TYPE st_OneDirectionCore :
STRUCT
  fname:STRING;
  index:LREAL;
  TargetDistance:LREAL;
  Execute:BOOL;
  Done:BOOL;
END_STRUCT
END_TYPE

(* stored: Version 1.1.0.1, ProductVersion 3.1.4024.13
   DUT st_OneDirectionCore: Id {bc800f46-fa73-4ac1-80a8-add29173b840} *)
